FUNCTION_BLOCK "Convention23"
TITLE = Test for rule Convention 23
VAR
bla : Any; // OK
END_VAR
BEGIN
END_FUNCTION_BLOCK
